// SIMATIC S7-200 project (STEP 7-Micro/WIN), CPU 224 CN REL 02.01

SYMBOL_TABLE 用户定义1
清仓               M0.4
电机故障             I0.1
换料               I0.0
取样周期             VW32
全部暂停             M0.3
手动报警             M10.3
手动自动             M0.2
换矿               M0.0
手卸料              M10.2
手开搅拌机            M10.1
手动开接料阀           M10.0
报警器              Q0.3
卸料阀              Q0.2
搅拌机              Q0.1
接料气动阀            Q0.0
END_SYMBOL_TABLE

ORGANIZATION_BLOCK 主程序:OB1
TITLE=程序注释
BEGIN
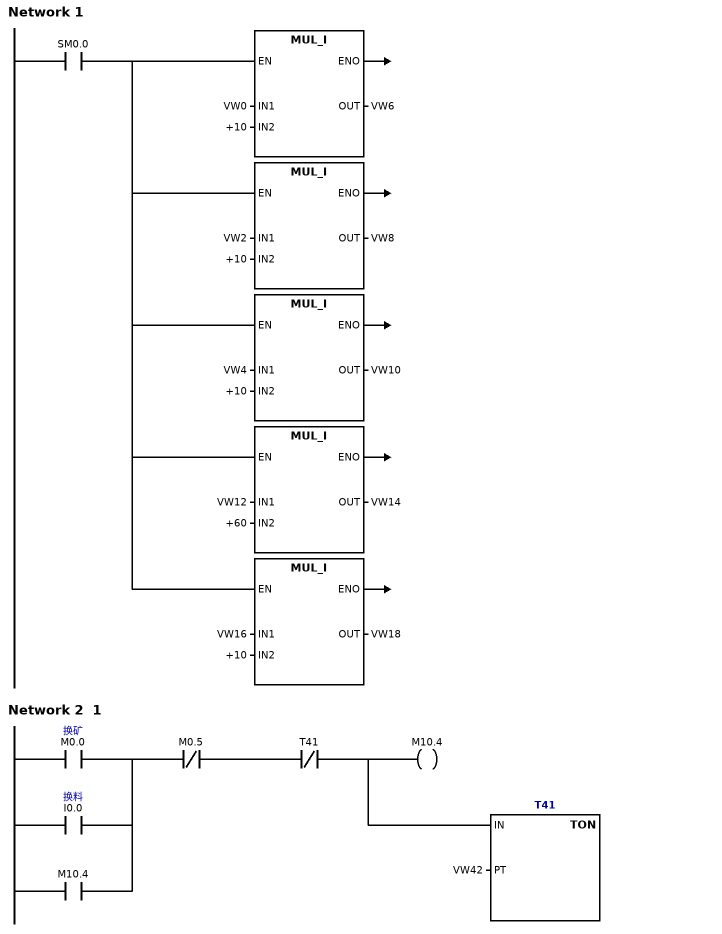
Network 1
LD     SM0.0
MOVW   VW0, VW6
*I     +10, VW6
MOVW   VW2, VW8
*I     +10, VW8
MOVW   VW4, VW10
*I     +10, VW10
MOVW   VW12, VW14
*I     +60, VW14
MOVW   VW16, VW18
*I     +10, VW18
Network 2 // 1
LD     换矿:M0.0
O      换料:I0.0
O      M10.4
AN     M0.5
AN     T41
=      M10.4
TON    T41, VW42
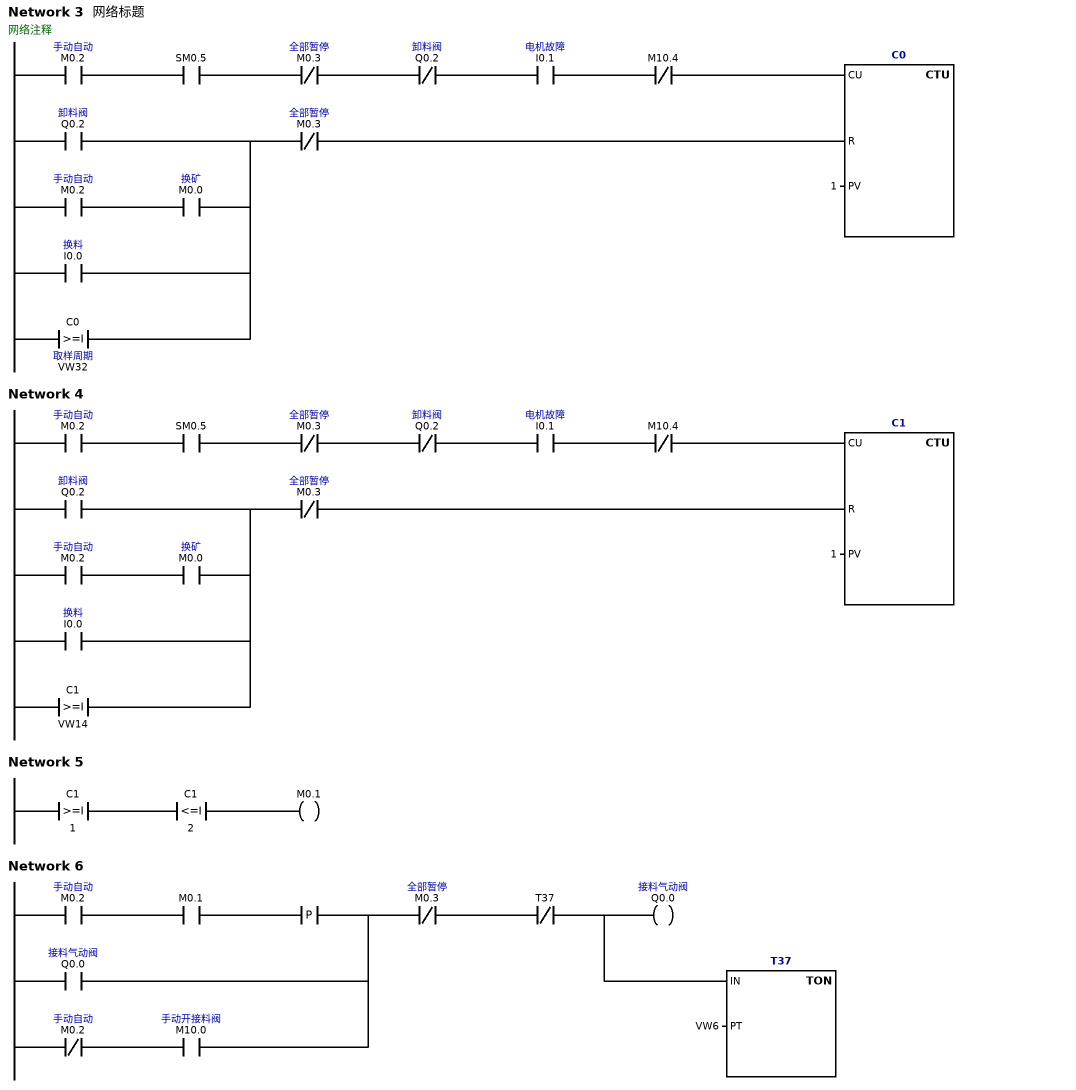
Network 3 // 网络标题
// 网络注释
LD     手动自动:M0.2
A      SM0.5
AN     全部暂停:M0.3
AN     卸料阀:Q0.2
A      电机故障:I0.1
AN     M10.4
LD     卸料阀:Q0.2
LD     手动自动:M0.2
A      换矿:M0.0
OLD
O      换料:I0.0
OW>=   C0, 取样周期:VW32
AN     全部暂停:M0.3
CTU    C0, 1
Network 4
LD     手动自动:M0.2
A      SM0.5
AN     全部暂停:M0.3
AN     卸料阀:Q0.2
A      电机故障:I0.1
AN     M10.4
LD     卸料阀:Q0.2
LD     手动自动:M0.2
A      换矿:M0.0
OLD
O      换料:I0.0
OW>=   C1, VW14
AN     全部暂停:M0.3
CTU    C1, 1
Network 5
LDW>=  C1, 1
AW<=   C1, 2
=      M0.1
Network 6
LD     手动自动:M0.2
A      M0.1
EU
O      接料气动阀:Q0.0
LDN    手动自动:M0.2
A      手动开接料阀:M10.0
OLD
AN     全部暂停:M0.3
AN     T37
=      接料气动阀:Q0.0
TON    T37, VW6
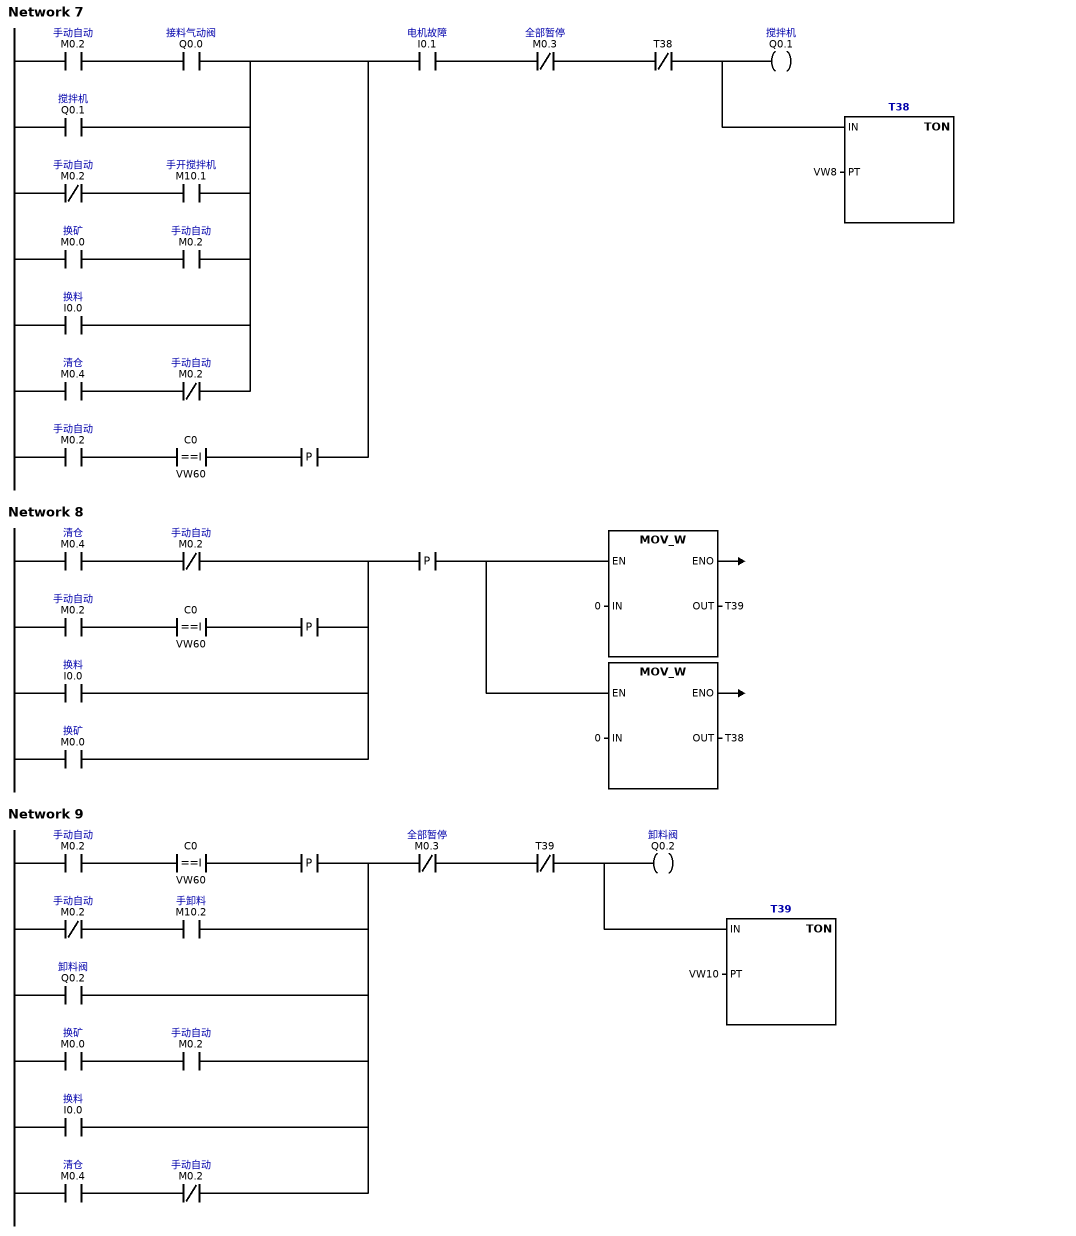
Network 7
LD     手动自动:M0.2
A      接料气动阀:Q0.0
O      搅拌机:Q0.1
LDN    手动自动:M0.2
A      手开搅拌机:M10.1
OLD
LD     换矿:M0.0
A      手动自动:M0.2
OLD
O      换料:I0.0
LD     清仓:M0.4
AN     手动自动:M0.2
OLD
LD     手动自动:M0.2
AW=    C0, VW60
EU
OLD
A      电机故障:I0.1
AN     全部暂停:M0.3
AN     T38
=      搅拌机:Q0.1
TON    T38, VW8
Network 8
LD     清仓:M0.4
AN     手动自动:M0.2
LD     手动自动:M0.2
AW=    C0, VW60
EU
OLD
O      换料:I0.0
O      换矿:M0.0
EU
MOVW   0, T39
MOVW   0, T38
Network 9
LD     手动自动:M0.2
AW=    C0, VW60
EU
LDN    手动自动:M0.2
A      手卸料:M10.2
OLD
O      卸料阀:Q0.2
LD     换矿:M0.0
A      手动自动:M0.2
OLD
O      换料:I0.0
LD     清仓:M0.4
AN     手动自动:M0.2
OLD
AN     全部暂停:M0.3
AN     T39
=      卸料阀:Q0.2
TON    T39, VW10
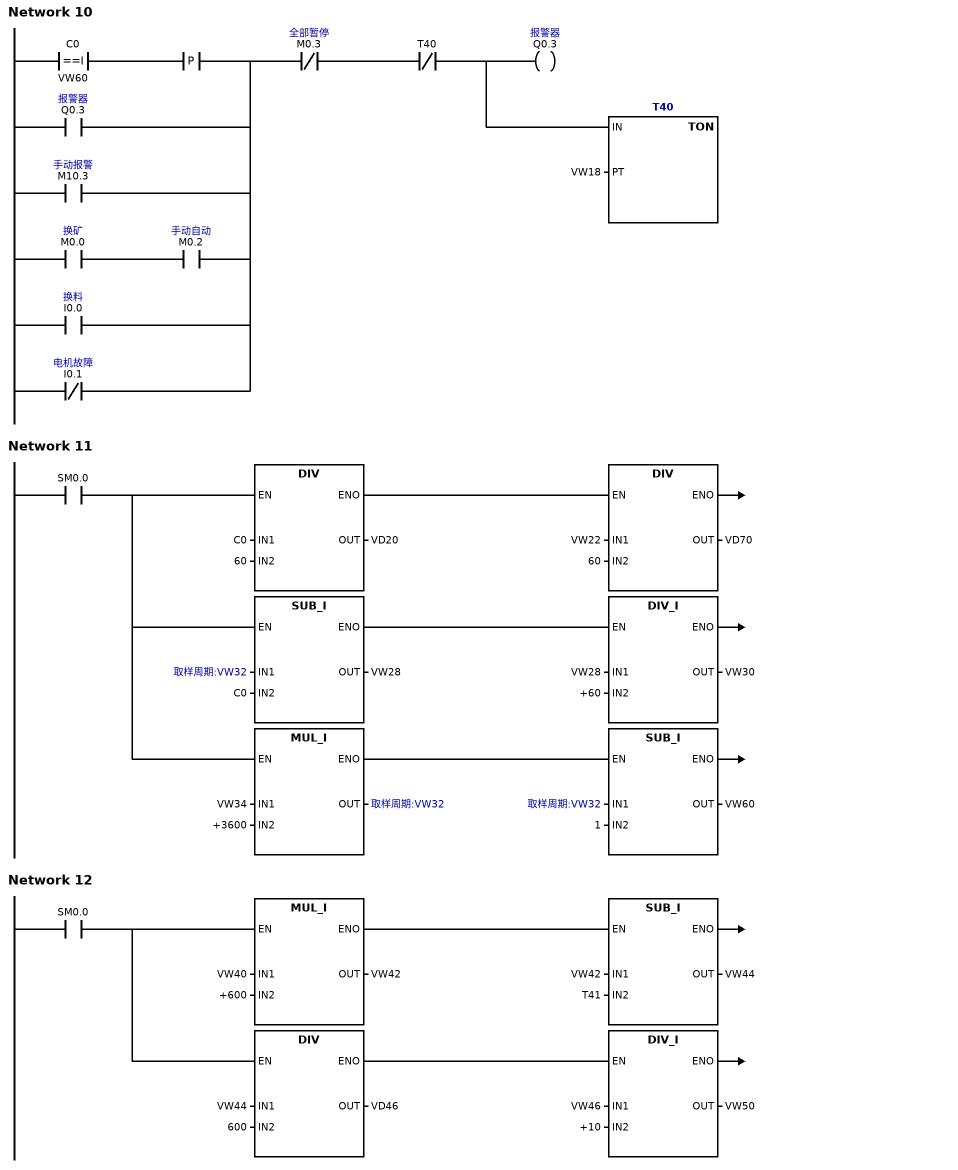
Network 10
LDW=   C0, VW60
EU
O      报警器:Q0.3
O      手动报警:M10.3
LD     换矿:M0.0
A      手动自动:M0.2
OLD
O      换料:I0.0
ON     电机故障:I0.1
AN     全部暂停:M0.3
AN     T40
=      报警器:Q0.3
TON    T40, VW18
Network 11
LD     SM0.0
LPS
MOVW   C0, VW22
AENO
DIV    60, VD20
AENO
MOVW   VW22, VW72
DIV    60, VD70
LRD
MOVW   取样周期:VW32, VW28
AENO
-I     C0, VW28
AENO
MOVW   VW28, VW30
/I     +60, VW30
LPP
MOVW   VW34, 取样周期:VW32
AENO
*I     +3600, 取样周期:VW32
AENO
MOVW   取样周期:VW32, VW60
-I     1, VW60
Network 12
LD     SM0.0
LPS
MOVW   VW40, VW42
AENO
*I     +600, VW42
AENO
MOVW   VW42, VW44
-I     T41, VW44
LPP
MOVW   VW44, VW48
AENO
DIV    600, VD46
AENO
MOVW   VW46, VW50
/I     +10, VW50
END_ORGANIZATION_BLOCK
